(* CODESYS project CtaAppSupperheat_2.0.0.0.library
   Description: Überhitzungsregelungs- Library der CTA
   Version: 2.0.0.0
   Title: CtaAppSuperheat
   Author: SIS
   DocFormat: reStructuredText
   Placeholder: CtaAppSuperheat
   LanguageModelAttribute: qualified-access-only
   DefaultNamespace: CtaAppSuperheat
   CompiledLibraryCompatibilityVersion: CODESYS V3.5 SP16 Patch 3
   Company: CTA

Project tree, tasks and I/O mapping:
  libraries: Standard, 3.5.18.0 (System); CtaSysConfig, 2.0.0.0 (CTA); CtaVisSymbols, 2.0.0.0 (CTA); VisuDialogs, 3.5.16.20 (System); VisuSymbols, 4.5.0.0 (System); CtaAppReport, 2.0.0.0 (CTA); CtaAppDumper, 2.0.0.0 (CTA); CtaAppPid, 2.0.0.0 (CTA); CtaAppFilter, 1.0.0.0 (CTA); CtaAppBasic, 1.0.0.0 (CTA); CtaAppBmk, 2.0.0.0 (CTA); CtaAppInfluxLog, 1.0.0.1 (CTA); CtaVisHelp, 2.0.0.0 (CTA)
  40 Visualizations/
    Report/
      visualisation ReportIcon
      visualisation VIS_SUPERHEAT_REPORTS
    Settings/
      visualisation VIS_SUPERHEAT_SETTINGS
      visualisation VIS_SUPERHEAT_SETTINGS_BASE
    PopUp/
      visualisation PopUp
    VisSuperheat/
      visualisation visSuperheat
  00000000-0000-0000-0000-000000000000|D:\CoDeSys\LibrariesV3\trunk\Intern\CAA\CAA Template\3.4.0.0 draft\Placeholder.xml
  00000000-0000-0000-0000-000000000000|D:\CoDeSys\LibrariesV3\trunk\Intern\CAA\CAA Template\3.2.0.3 draft\Prefix.pdf
  00000000-0000-0000-0000-000000000000|D:\CoDeSys\LibrariesV3\trunk\Intern\CAA\CAA Template\3.5.2.0 draft\Placeholder.xml
  20 Structs/
    data type scParameter
    BASE/
      data type scBase
    InfluxDb/
      data type scInfluxDb
    LowSuperheat/
      data type scLowSuperheat
    MOP/
      data type scMOP
    Manual/
      data type scManual
  50 Images/
  10 Documenation/
    global variables VersionHistory
    global variables readMe
  21 Interface/
    interface ITF_Superheat: proAcknowleg, proAvailable, proLockDown, proIsError, proIsWarning, prorOnY, prorLowSuperheatValue, prorActÜberhitzung, prorSollÜberhitzung, p_scBase_fbxEnable, p_scBase_EnAlarmVentOffen, p_scBase_fbtDelayStartAlarm, p_scInfluxDb_fbxEnable, p_scLowSuperheat_fbrMin, p_scLowSuperheat_fbxEnable, p_scLowSuperheat_fbtDelayStartRegler, p_scLowSuperheat_fbrMax, p_scLowSuperheat_fbrMinÖffnung, p_scLowSuperheat_fbxEnableWarning, p_scLowSuperheat_fbxEnableAlarm, p_scLowSuperheat_fbtDelayStartAlarm, P_scLowSuperheat_fbrLowShAlarmValue, p_scMOP_fbxEnable, p_scMOP_fbxEnableWarning, p_scMOP_fbxEnableAlarm, p_scMOP_fbtDelayStartAlarm, p_scMOP_fbrMopSollwert, proRefTofbPidSuperheat, proRefTofbSuperheatDumper, proRefTofbPidMop, proRefTofbMopDumper, proITF_REPORTMANAGER
  11 Library Parameter/
  12 Konstanten/
    global variables GlobalKonstant
  60 Textlisten/
    text list Error
    text list Info
    text list Warnung
  13 Globale Variablen/
  text list GlobalTextList
  5ce3da45-db07-42e7-a21c-a00fff4ed8f6|C:\Users\sis\Downloads\dip-switch.svg
  5ce3da45-db07-42e7-a21c-a00fff4ed8f6|C:\Users\sis\Downloads\lightning-bolt-circle.svg
  30 Program Organization Units/
    function block fbSuperheat [ST]: actConfigFile, actReport, actTrendlog, actState, prorOnY, prorActÜberhitzung, prorLowSuperheatValue, prorSollÜberhitzung, proITF_REPORTMANAGER, proAcknowleg, proAvailable, proLockDown, proIsWarning, proIsError, p_scMOP_fbxEnable, p_scMOP_fbxEnableWarning, p_scMOP_fbxEnableAlarm, p_scMOP_fbtDelayStartAlarm, p_scMOP_fbrMopSollwert, p_scManual_fbxEnable, p_scManual_fbrManualValue, p_scInfluxDb_fbxEnable, p_scLowSuperheat_fbtDelayStartRegler, p_scLowSuperheat_fbrMin, p_scLowSuperheat_fbrMax, p_scLowSuperheat_fbrMinÖffnung, p_scLowSuperheat_fbxEnableWarning, p_scLowSuperheat_fbxEnableAlarm, p_scLowSuperheat_fbtDelayStartAlarm, p_scLowSuperheat_fbxEnable, P_scLowSuperheat_fbrLowShAlarmValue, p_scBase_fbxEnable, p_scBase_EnAlarmVentOffen, p_scBase_fbtDelayStartAlarm, proRefTofbPidSuperheat, proRefTofbSuperheatDumper, proRefTofbPidMop, proRefTofbMopDumper
    function fcProcentualReduction [ST]
  5ce3da45-db07-42e7-a21c-a00fff4ed8f6|C:\Users\sis\Downloads\sine-wave.svg
  5ce3da45-db07-42e7-a21c-a00fff4ed8f6|C:\Users\sis\Downloads\eye.svg
  5ce3da45-db07-42e7-a21c-a00fff4ed8f6|C:\Users\sis\Downloads\lan.svg
*)

// 20 Structs/scParameter
{attribute 'pack_mode' := '1'} 
TYPE scParameter :
	STRUCT
		scBase			: 	scBase;
		scLowSuperheat	:	scLowSuperheat;
		scMOP			:	scMOP;
		scManual		:	scManual;
		scInfluxDb		:	scInfluxDb;
	END_STRUCT
END_TYPE

// 20 Structs/BASE/scBase
TYPE scBase :
	STRUCT	
		fbxEnable				:	CtaSysConfig.fbBOOL;
		fbxEnAlarmVentOffen		:	CtaSysConfig.fbBOOL;
		fbtDelayStartAlarm		:	CtaSysConfig.fbTIME;		
	END_STRUCT
END_TYPE

// 20 Structs/InfluxDb/scInfluxDb
TYPE scInfluxDb :
	STRUCT		
		fbxEnable			:	CtaSysConfig.fbBOOL;
	END_STRUCT
END_TYPE

// 20 Structs/LowSuperheat/scLowSuperheat
TYPE scLowSuperheat :
	STRUCT
		fbxEnable				:	CtaSysConfig.fbBOOL;
		fbtDelayStartRegler		:	CtaSysConfig.fbTIME;
		fbrMin					:	CtaSysConfig.fbREAL;
		fbrMax					:	CtaSysConfig.fbREAL;
		fbrMinÖffnung			:	CtaSysConfig.fbREAL;
		fbxEnableWarning		:	CtaSysConfig.fbBOOL;
		fbxEnableAlarm			:	CtaSysConfig.fbBOOL;
		fbtDelayStartAlarm		:	CtaSysConfig.fbTIME;
		fbrLowShAlarmValue		:	CtaSysConfig.fbREAL;
	END_STRUCT
END_TYPE

// 20 Structs/MOP/scMOP
TYPE scMOP :
	STRUCT
		fbxEnable				:	CtaSysConfig.fbBOOL;
		fbxEnableWarning		:	CtaSysConfig.fbBOOL;
		fbxEnableAlarm			:	CtaSysConfig.fbBOOL;
		fbtDelayStartAlarm		:	CtaSysConfig.fbTIME;
		fbrMopSollwert			:	CtaSysConfig.fbREAL;
	END_STRUCT
END_TYPE

// 20 Structs/Manual/scManual
TYPE scManual :
	STRUCT
		fbxEnable		: CtaSysConfig.fbBOOL;
		fbrManualValue	: CtaSysConfig.fbREAL;
	END_STRUCT
END_TYPE

// 10 Documenation/VersionHistory
(* 

.. image:: ../../Images/CTA_Logo.jpg
   :align: right
   :width: 15% 

**Vorlage**   


============ =========== =========== ============================================
**Date**     **Version** **Author**  **Change**
------------ ----------- ----------- --------------------------------------------
04.03.2021   0.0.0.0     SIS         Vorlage erstellt

============ =========== =========== ============================================


*)
VAR_GLOBAL
    stInfo : STRING:= '0.0.0.0, Vorlage, CTA';
END_VAR

// 10 Documenation/readMe
(*

**ReadMe**
 
|	**Empfehlung**
|
|	Die Bibliothek CtaAppSuperheat dient der Überhitzungsregelung und errechnet den Stellwert für das elektronische Einspritzventil.
|	Instanzieren Sie den CtaAppSuperheat.fbSuperheat in ihrem Funktionsbaustein oder POU beispielsweise als fbSuperheatCtrl oder beliebig.
|	Deklarieren Sie die Struktur Variable welche als Parameter und zur ansteuerung dienen wie im Code beispiel.
|  
| *Beispiel* 

+-----------------------+---------------------------------------------------------------------------------------------------------------------------------------------------------------------------------------------------------------------------------------------------------------------------------------------------------------------------------------------------------------------------------------------------------------------------------------+
| Beschreibung          |  Code                                                                                                                                                                                                                                                                                                                                                                                                                                 |
+=======================+=======================================================================================================================================================================================================================================================================================================================================================================================================================================+
| Pou oder SmFb         | .. code-block:: codesys                                                                                                                                                                                                                                                                                                                                                                                                               |
|                       |                                                                                                                                                                                                                                                                                                                                                                                                                                       |
|                       |	// Deklaration als VAR im POU oder dem selbsterstellten Funktionsbaustein                                                                                                                                                                                                                                                                                                                                                       	|
|                       |   VAR   																																																																																																								|
|						|	    (*Überhitzungsregelung*)																																																		 																																																|
|						|		fbSuperheatCtrl			: CtaAppSuperheat.fbSuperheat;                                                                                                                                                                                                                                                                                                                                                             				|
|						|																																																																																																										|
+-----------------------+---------------------------------------------------------------------------------------------------------------------------------------------------------------------------------------------------------------------------------------------------------------------------------------------------------------------------------------------------------------------------------------------------------------------------------------+
| Code für Init         | .. code-block:: codesys                                                                                                                                                                                                                                                                                                                                                                                                               |
|                       |   																																																																																																									|
| 						|	// Kopieren des nachfolgenden Codes in eine Action zur Initialisierung der Parameter. Zum Beispiel actConfig.																																																																														|
|                       |	{region "Überhitzungsregelung																																																																																																		|
|						|		(*Base*)                                                                                                                                                                                                                                                                                                                                                                                                   						|
|						|		fbSuperheatCtrl.scParameter.scBase.fbxEnable						(_wertInit :=	 TRUE														);		//P1 Überhitzungsregelung aktiv / inaktiv																																																								|
|						|		fbSuperheatCtrl.scParameter.scBase.fbrStartÖffnung					(_wertInit :=	   20		, _minInit :=			, _maxInit :=			);		//P2 Startöffnung des Ventils																																																											|
|						|		fbSuperheatCtrl.scParameter.scBase.fbtDelayStartRegler				(_wertInit :=	T#10s		, _minInit :=			, _maxInit :=			);		//P3 Startverzögerung der Regelung																																																										|
|						|		fbSuperheatCtrl.scParameter.scBase.fbxEnAlarmVentOffen				(_wertInit :=	FALSE														);		//P4 Alarm bei 100% geöffnetem Ventil aktiv / inaktiv																																																					|
|						|		fbSuperheatCtrl.scParameter.scBase.fbtDelayStartAlarm				(_wertInit :=	 T#0S		, _minInit :=			, _maxInit :=			);		//P5 Alarmverzögerung 																																																													|
|						|																																																																																																										|
|						|		(*Superheat PID*)																																																																																																				|
|						|		fbSuperheatCtrl.fbPidSuperheat.scParameter.fbrBand					(_wertInit :=	   15		, _minInit :=			, _maxInit :=			);		//P6  Superheat PID - Band																																																												|
|						|		fbSuperheatCtrl.fbPidSuperheat.scParameter.fbrDeadBand				(_wertInit :=	 0.10		, _minInit :=			, _maxInit :=			);		//P7  Superheat PID - Totband																																																											|
|						|		fbSuperheatCtrl.fbPidSuperheat.scParameter.fbrTn					(_wertInit :=	   25		, _minInit :=			, _maxInit :=			);		//P8  Superheat PID - I Anteil																																																											|
|						|		fbSuperheatCtrl.fbPidSuperheat.scParameter.fbrTv					(_wertInit :=	    2		, _minInit :=			, _maxInit :=			);		//P9  Superheat PID - D Anteil																																																											|
|						|		fbSuperheatCtrl.fbPidSuperheat.scParameter.fbxEnTrendlog			(_wertInit :=	FALSE														);		//P10 Superheat PID - Trendaufzeichnung																																																									|
|						|		fbSuperheatCtrl.fbPidSuperheat.scParameter.fbxInvert				(_wertInit :=	FALSE														);		//P11 Superheat PID - Invrtierung																																																										|
|						|																																																																																																										|
|						|		(*Superheat Dumper*)																																																																																																			|
|						|		fbSuperheatCtrl.fbSuperheatDumper.scParameter.fbrBand				(_wertInit :=	  100		, _minInit :=			, _maxInit :=			);		//P12 Superheat Dumper - Band																																																											|
|						|		fbSuperheatCtrl.fbSuperheatDumper.scParameter.fbrTup				(_wertInit :=	   10		, _minInit :=			, _maxInit :=			);		//P13 Superheat Dumper - Zuschaltzeit																																																									|
|						|		fbSuperheatCtrl.fbSuperheatDumper.scParameter.fbrTdown				(_wertInit :=	    1		, _minInit :=			, _maxInit :=			);		//P14 Superheat Dumper - Wegschaltzeit																																																									|
|						|		fbSuperheatCtrl.fbSuperheatDumper.scParameter.fbxInExpOut			(_wertInit :=	FALSE														);		//P15 Superheat Dumper - In = Out annahme																																																								|
|						|																																																																																																										|
|						|		(*Low Superheat*)																																																																																																				|
|						|		fbSuperheatCtrl.scParameter.scLowSuperheat.fbxEnable				(_wertInit :=	 TRUE														);		//P16 LowSuperheat aktiv / inaktiv																																																										|
|						|		fbSuperheatCtrl.scParameter.scLowSuperheat.fbrMin					(_wertInit :=	  2.0		, _minInit :=			, _maxInit :=			);		//P17 LowSuperheat Minimalwert																																																											|
|						|		fbSuperheatCtrl.scParameter.scLowSuperheat.fbrMax					(_wertInit :=	  3.0		, _minInit :=			, _maxInit :=			);		//P18 LowSuperheat Maximalwert																																																											|
|						|		fbSuperheatCtrl.scParameter.scLowSuperheat.fbrMinÖffnung			(_wertInit :=	 	0		, _minInit :=			, _maxInit :=			);		//P19 LowSuperheat Minimalöffnung																																																										|
|						|		fbSuperheatCtrl.scParameter.scLowSuperheat.fbtDelayStartRegler		(_wertInit :=	T#30s		, _minInit :=			, _maxInit :=			);		//P20 LowSuperheat Regler Startverzögerung																																																								|
|						|		fbSuperheatCtrl.scParameter.scLowSuperheat.fbxEnableWarning			(_wertInit :=	 TRUE														);		//P21 LowSuperheat Warnung aktiv / inaktiv																																																								|
|						|		fbSuperheatCtrl.scParameter.scLowSuperheat.fbxEnableAlarm			(_wertInit :=	 TRUE														);		//P22 LowSuperheat Alarm aktiv / inaktiv																																																								|
|						|		fbSuperheatCtrl.scParameter.scLowSuperheat.fbtDelayStartAlarm		(_wertInit :=	T#30s		, _minInit :=			, _maxInit :=			);		//P23 LowSuperheat Alarmverzögerung																																																										|
|						|																																																																																																										|
|						|		(*MOP*)																																																																																																							|
|						|		fbSuperheatCtrl.scParameter.scMOP.fbxEnable							(_wertInit :=	 TRUE														);		//P24 MOP aktiv / inaktiv																																																												|
|						|		fbSuperheatCtrl.scParameter.scMOP.fbxEnableWarning					(_wertInit :=	 TRUE														);		//P25 MOP Warnung aktiv / inaktiv																																																										|
|						|		fbSuperheatCtrl.scParameter.scMOP.fbxEnableAlarm					(_wertInit :=	 TRUE														);		//P26 MOP Alarm aktiv / inaktiv																																																											|
|						|		fbSuperheatCtrl.scParameter.scMOP.fbtDelayStartAlarm				(_wertInit :=	T#10s		, _minInit :=			, _maxInit :=			);		//P27 MOP Alarmverzögerung																																																												|
|						|																																																																																																										|
|						|		(*MOP Leistungsreduktion*)																																																																																																		|
|						|		fbSuperheatCtrl.fbMopLeistungsreduktion.scParameter.fbxEn			(_wertInit :=	 TRUE														);		//P28 MOP Leistungsreduktion aktiv / inaktiv 																																																							|
|						|		fbSuperheatCtrl.fbMopLeistungsreduktion.scParameter.fbtStartTime	(_wertInit :=	 T#1m		, _minInit :=			, _maxInit :=			);		//P29 MOP Leistungsreduktion Regler Startverzögerung																																																					|
|						|		fbSuperheatCtrl.fbMopLeistungsreduktion.scParameter.fbtRunTime		(_wertInit :=	 T#1m		, _minInit :=			, _maxInit :=			);		//P30 MOP Leistungsreduktion Regler Betriebsverzögerung																																																					|
|						|		fbSuperheatCtrl.fbMopLeistungsreduktion.scParameter.fbrSoll			(_wertInit :=	   10		, _minInit :=			, _maxInit :=			);		//P31 MOP Leistungsreduktion Sollwert																																																									|
|						|		fbSuperheatCtrl.fbMopLeistungsreduktion.scParameter.fbrCounter		(_wertInit :=	 	5		, _minInit :=			, _maxInit :=			);		//P32 MOP Leistungsreduktion Weg- / Zuschaltungwert																																																						|
|						|		fbSuperheatCtrl.fbMopLeistungsreduktion.scParameter.fbxEnTrendLog	(_wertInit :=	 TRUE														);		//P33 MOP Leistungsreduktion Trendaufzeichnung																																																							|
|						|																																																																																																										|
|						|		(*MOP Dumper*)																																																																																																					|
|						|		fbSuperheatCtrl.fbMopDumper.scParameter.fbrBand						(_wertInit :=	  0.0		, _minInit :=			, _maxInit :=			);		//P34 MOP Dumper - Band																																																													|
|						|		fbSuperheatCtrl.fbMopDumper.scParameter.fbrTdown					(_wertInit :=	 0.10		, _minInit :=			, _maxInit :=			);		//P35 MOP Dumper - Zuschaltzeit																																																											|
|						|		fbSuperheatCtrl.fbMopDumper.scParameter.fbrTup						(_wertInit :=	 0.10		, _minInit :=			, _maxInit :=			);		//P36 MOP Dumper - Wegschaltzeit																																																										|
|						|		fbSuperheatCtrl.fbMopDumper.scParameter.fbxInExpOut					(_wertInit :=	FALSE														);		//P37 MOP In = Out annahme																																																												|
|						|																																																																																																										|
|						|		(*Manual*)																																																																																																						|
|						|		fbSuperheatCtrl.scParameter.scManual.fbxEnable						(_wertInit :=	FALSE														);		//P38 Manuelle Übersteuerung aktivieren / deaktivieren																																																					|
|						|		fbSuperheatCtrl.scParameter.scManual.fbrManualValue					(_wertInit :=	 	0		, _minInit :=			, _maxInit :=			);		//P39 Manueller Ventilstellwert																																																											|
|						|																																																																																																										|
|						|		(*Trendlog*)																																																																																																					|
|						|		fbSuperheatCtrl.scParameter.scInfluxDb.fbxEnable					(_wertInit :=	 TRUE														);		//P40 Überhitzungsregelung Trendaufzeichnung																																																							|
|						|	{endregion}                                                                                                                                                      																																																																	|
+-----------------------+---------------------------------------------------------------------------------------------------------------------------------------------------------------------------------------------------------------------------------------------------------------------------------------------------------------------------------------------------------------------------------------------------------------------------------------+
*)                                                                                                                                                                                                                                                                                                                                                                                                                                                               
 VAR_GLOBAL                                                                                                                                                                                                                                                                                                                                                                                                                                                      
    xReadMeDone              :   BOOL;                                                                                                                                                                                                                                                                                                                                                                                                                           
END_VAR

// 12 Konstanten/GlobalKonstant
{attribute 'qualified_only'}
VAR_GLOBAL
	stReportTextListError   : CtaAppReport.stReportTextList := 'CtaAppSuperheat.Error';
	stReportTextListWarning : CtaAppReport.stReportTextList := 'CtaAppSuperheat.Warnung';
	stReportTextListInfo    : CtaAppReport.stReportTextList := 'CtaAppSuperheat.Info';	
END_VAR

// 30 Program Organization Units/fbSuperheat
FUNCTION_BLOCK fbSuperheat IMPLEMENTS ITF_Superheat
VAR_INPUT
	
	//Überhitzungsregler   
    xRelease						: BOOL;	// Freigabe Regulierung, Beispiel Freigabe Verdichter
    rSollÜberhitzung				: REAL;	// Sollwert Überhitzung
    rKorrekturÜberhizungssollwert	: REAL;	// Korrektur von Sollwert, Schiebungswert muss aussen gemacht werden
    rActSauggastemperatur			: REAL;
    rActVerdampfungstemperatur		: REAL;
	ITF_BMK							: CtaAppBmk.ITF_BMK;
	
END_VAR
VAR_OUTPUT
	 rOnY							: REAL;	// Aktueller Stellwert für Expansionsventil
END_VAR
VAR
	(* Internal States *) 
	scEWI							: CtaAppReport.scReportNr;
	_xIsWarning						: BOOL;
	xIsWarning						: BOOL;
	_xIsError						: BOOL;
	xIsError						: BOOL;
	xisEnabled						: BOOL;
		
	(* Temps and Helpers *)
	rLowSuperheatScaled				: REAL;
	xConfigError					: BOOL;
	
	(* Bausteine Superheat *)	
	fbPidSuperheat					: CtaAppPid.fbPid;
	fbSuperheatDumper				: CtaAppDumper.fbDumper;
	
	(* Bausteine Low Superheat *)
	fbLowSuperheatDelay				: Standard.TON;
	fbLowSuperheatSetReset			: Standard.RS;
	fbLowSuperheatFilter			: CtaAppFilter.fbImpulsFilter;
	
	(* Bausteine MOP *)
	fbPidMop						: CtaAppPid.fbPid;
	fbMopDumper						: CtaAppDumper.fbDumper;
	
	(* Reporting *) 
	fbReportManager			    	: CtaAppReport.fbReportManager;      
    difor					    	: DINT;                                                                    
    ayErrorReporter					: ARRAY[1..5] OF CtaAppReport.fbReporter;
	ayWarningReporter				: ARRAY[1..2] OF CtaAppReport.fbReporter;
	
	(* Trendlogs *)
	fbTrendxOn						:	CtaAppInfluxLog.FB_LOG_NODE_BOOL;
	fbTrendrOny						:	CtaAppInfluxLog.FB_LOG_NODE_REAL;
	fbTrendxWarning					:	CtaAppInfluxLog.FB_LOG_NODE_BOOL;
	fbTrendxError					:	CtaAppInfluxLog.FB_LOG_NODE_BOOL;
	(* ConfigFile *)
	fbConfigfile					: CtaSysConfig.fbConfigFile;
	scParameter						: scParameter;
END_VAR

actConfigFile();

IF xIsEnabled AND NOT xConfigError THEN
	
	(* Superheat *)
	
		// PID
		fbPidSuperheat(	xEn 					:=	xRelease,
						rAct 					:=	rActSauggastemperatur - rActVerdampfungstemperatur,
						rSoll 					:=	rSollÜberhitzung + rKorrekturÜberhizungssollwert,
						stPhysikalischeEinheit 	:=	'°c');
						
		// Skalierung 			
		fbSuperheatDumper.rSoll :=  CtaAppBasic.fcScale(rIn 	:= fbPidSuperheat.rY,
														rMin 	:=	-100,
														rMax 	:=	 100,
														rOutMin	:=	   0,
														rOutMax	:=   100);
		// Dämpfung des skalierten Wertes												
		fbSuperheatDumper(xEn := TRUE);				
	
	(* Low Superheat *)
		// Skalierung
		rLowSuperheatScaled := MAX (0 , CtaAppBasic.fcScale(rIn 	:= fbPidSuperheat.rAct,
															rMin 	:= scParameter.scLowSuperheat.fbrMin.proValue,
															rMax 	:= scParameter.scLowSuperheat.fbrMax.proValue,
															rOutMin := 100 - scParameter.scLowSuperheat.fbrMinÖffnung.proValue,
															rOutMax := 0));
		
		// Verzögerung der Regelung
		fbLowSuperheatDelay(IN :=	xRelease 										AND
									(rLowSuperheatScaled > 0) 						AND 
								 	NOT fbLowSuperheatSetReset.Q1 					AND
								  	scParameter.scLowSuperheat.fbxEnable.proValue,
							PT := 	scParameter.scLowSuperheat.fbtDelayStartRegler.proValue);
							
		// Set Reset					
		fbLowSuperheatSetReset(	SET 	:= fbLowSuperheatDelay.Q ,
								RESET1 	:= NOT xRelease);
		
		// Wert für prozentuale Reduktion LowSuperheat				
		IF fbLowSuperheatSetReset.Q1 THEN
			fbLowSuperheatFilter.rIn := rLowSuperheatScaled;
		ELSE
			fbLowSuperheatFilter.rIn := 0;
		END_IF
		
		// Filterung des Wertes
		fbLowSuperheatFilter(rFilter := 10.0);
		
		// LowSuperheat reporting in der Aktion actReport realisiert
	
	(* MOP *)
		// Leistungreduktion
		fbPidMop(	xEn 					:= xRelease AND scParameter.scMOP.fbxEnable.proValue,
					rAct 					:= rActVerdampfungstemperatur,
					rSoll 					:= scParameter.scMOP.fbrMopSollwert.proValue,
					stPhysikalischeEinheit 	:= '°c'  );
								
		// Dämpfung des MOP- Wertes
		fbMopDumper(xEn 	:= xRelease AND scParameter.scMOP.fbxEnable.proValue,
					rSoll 	:= LIMIT(0,fbPidMop.rY,100));
		
		// MOP Reporting in der Aktion actReport realisiert
	
	(* Stellwert *)
	IF xRelease THEN
		// Ausgang mit prozentualer Reduktion beschalten
		fcProcentualReduction(	rLAkt 	:= fbSuperheatDumper.rY,
								rLR1	:= fbLowSuperheatFilter.rOut,
								rLR2	:= fbMopDumper.rY,
								rOut	=> rOnY);		
	ELSE
		rOnY := 0;	
	END_IF	
	
	// Reports
	IF __QUERYINTERFACE(ITF_BMK,ITF_BMK)THEN
		actReport();
	END_IF
ELSE
	// Stellwertreporting in der Atkion actReport realisiert
	rOnY := 0;
	
	// Konfigurationsfehler
	IF xConfigError THEN
		IF __QUERYINTERFACE(ITF_BMK,ITF_BMK)THEN
			actReport();
		END_IF
	END_IF	
END_IF

// Status
actState();
// Trends
IF __QUERYINTERFACE(ITF_BMK,ITF_BMK) THEN
	actTrendlog();
END_IF

ACTION actConfigFile:
fbConfigfile();

(* Basisparameter *)
scParameter.scBase.fbxEnable					(_usiParaNr :=  1, ItfConfigFb := fbConfigFile);
scParameter.scBase.fbxEnAlarmVentOffen 			(_usiParaNr :=  4, ItfConfigFb := fbConfigFile);
scParameter.scBase.fbtDelayStartAlarm			(_usiParaNr :=  5, ItfConfigFb := fbConfigFile);
(* Low Superheat *)
scParameter.scLowSuperheat.fbxEnable			(_usiParaNr :=  6, ItfConfigFb := fbConfigFile);
scParameter.scLowSuperheat.fbtDelayStartRegler	(_usiParaNr :=  7, ItfConfigFb := fbConfigFile);
scParameter.scLowSuperheat.fbrMin				(_usiParaNr :=  8, ItfConfigFb := fbConfigFile);
scParameter.scLowSuperheat.fbrMax				(_usiParaNr :=  9, ItfConfigFb := fbConfigFile);
scParameter.scLowSuperheat.fbrMinÖffnung		(_usiParaNr := 10, ItfConfigFb := fbConfigFile);
scParameter.scLowSuperheat.fbxEnableWarning		(_usiParaNr := 11, ItfConfigFb := fbConfigFile);
scParameter.scLowSuperheat.fbxEnableAlarm		(_usiParaNr := 12, ItfConfigFb := fbConfigFile);
scParameter.scLowSuperheat.fbtDelayStartAlarm	(_usiParaNr := 13, ItfConfigFb := fbConfigFile);
(* MOP Regler *)
scParameter.scMOP.fbxEnable						(_usiParaNr := 14, ItfConfigFb := fbConfigFile);
scParameter.scMOP.fbxEnableWarning				(_usiParaNr := 15, ItfConfigFb := fbConfigFile);
scParameter.scMOP.fbxEnableAlarm				(_usiParaNr := 16, ItfConfigFb := fbConfigFile);
scParameter.scMOP.fbtDelayStartAlarm			(_usiParaNr := 17, ItfConfigFb := fbConfigFile);
scParameter.scMOP.fbrMopSollwert				(_usiParaNr := 18, ItfConfigFb := fbConfigFile);
(* Trendlog *)
scParameter.scInfluxDb.fbxEnable				(_usiParaNr := 19, ItfConfigFb := fbConfigFile);

scParameter.scLowSuperheat.fbrLowShAlarmValue	(_usiParaNr := 20, ItfConfigFb := fbConfigFile);

xConfigError := fbConfigFile.xError;
END_ACTION

ACTION actReport:
(* EWI Manager *)
fbReportManager(	stErrorInitReportTextListIn		:=	ADR(GlobalKonstant.stReportTextListError),
					stWarningInitReportTextListIn	:=	ADR(GlobalKonstant.stReportTextListWarning),
					stInfoInitReportTextListIn		:=	ADR(GlobalKonstant.stReportTextListInfo),
					scReportNr						:=	scEWI);
					
(* Errors *)                        
        (* Meldung Error Low Superheat *)
        ayErrorReporter[1].proPrio  := 3;
        ayErrorReporter[1].metReport(     		xSetReportIn					:= xRelease AND 
																				   (rLowSuperheatScaled > 0) AND 
																				   scParameter.scLowSuperheat.fbxEnable.proValue AND
																				   scParameter.scLowSuperheat.fbxEnableAlarm.proValue,
												iReportID						:= 1,
												enReportTypeIn					:= CtaAppReport.enReportType.Error,  
												enReportAcknowledgeTypeIn   	:= CtaAppReport.enReportacknowledgeType.Quit,
												tDelay							:= scParameter.scLowSuperheat.fbtDelayStartAlarm.proValue, 
												ITF_BMK_IN						:= ITF_BMK,			              
												pstReportTextListIn				:= ADR(GlobalKonstant.stReportTextListError),
												stOptionalReportText		    := '',   
												iRetryTilReportLock 		    := 0, 
												xResetCount         		    := FALSE,  
												tReset						    := T#24H); 

		(* Meldung Error MOP *)
        ayErrorReporter[2].proPrio  := 3;
        ayErrorReporter[2].metReport(     		xSetReportIn					:= xRelease 			AND
																				   fbMopDumper.rY > 0 	AND 
																				   scParameter.scMOP.fbxEnableAlarm.proValue,
												iReportID						:= 2,
												enReportTypeIn					:= CtaAppReport.enReportType.Error,  
												enReportAcknowledgeTypeIn   	:= CtaAppReport.enReportacknowledgeType.Quit,
												tDelay							:= scParameter.scMOP.fbtDelayStartAlarm.proValue, 
												ITF_BMK_IN						:= ITF_BMK,			              
												pstReportTextListIn				:= ADR(GlobalKonstant.stReportTextListError),
												stOptionalReportText		    := '',   
												iRetryTilReportLock 		    := 0, 
												xResetCount         		    := FALSE,  
												tReset						    := T#24H);

		(* Meldung Error Ventil *)
        ayErrorReporter[3].proPrio  := 3;
        ayErrorReporter[3].metReport(     		xSetReportIn					:= (rOnY > 99.9) AND
																				   scParameter.scBase.fbxEnAlarmVentOffen.proValue,
												iReportID						:= 3,
												enReportTypeIn					:= CtaAppReport.enReportType.Error,  
												enReportAcknowledgeTypeIn   	:= CtaAppReport.enReportacknowledgeType.Quit,
												tDelay							:= scParameter.scBase.fbtDelayStartAlarm.proValue, 
												ITF_BMK_IN						:= ITF_BMK,			              
												pstReportTextListIn				:= ADR(GlobalKonstant.stReportTextListError),
												stOptionalReportText		    := '',   
												iRetryTilReportLock 		    := 0, 
												xResetCount         		    := FALSE,  
												tReset						    := T#24H);		
												
		(* Meldung Configerror *)
        ayErrorReporter[4].proPrio  := 1;
        ayErrorReporter[4].metReport(     		xSetReportIn					:= xConfigError,
												iReportID						:= 4,
												enReportTypeIn					:= CtaAppReport.enReportType.Error,  
												enReportAcknowledgeTypeIn   	:= CtaAppReport.enReportacknowledgeType.Quit,
												tDelay							:= scParameter.scBase.fbtDelayStartAlarm.proValue, 
												ITF_BMK_IN						:= ITF_BMK,			              
												pstReportTextListIn				:= ADR(GlobalKonstant.stReportTextListError),
												stOptionalReportText		    := '',   
												iRetryTilReportLock 		    := 0, 
												xResetCount         		    := FALSE,  
												tReset						    := T#24H);	

        (* Meldung Error Low Superheat *)
        ayErrorReporter[5].proPrio  := 1;
        ayErrorReporter[5].metReport(     		xSetReportIn					:= xRelease AND rActSauggastemperatur - rActVerdampfungstemperatur < scParameter.scLowSuperheat.fbrLowShAlarmValue.proValue,
												iReportID						:= 5,
												enReportTypeIn					:= CtaAppReport.enReportType.Error,  
												enReportAcknowledgeTypeIn   	:= CtaAppReport.enReportacknowledgeType.Quit,
												tDelay							:= T#1.5S, 
												ITF_BMK_IN						:= ITF_BMK,			              
												pstReportTextListIn				:= ADR(GlobalKonstant.stReportTextListError),
												stOptionalReportText		    := '',   
												iRetryTilReportLock 		    := 0, 
												xResetCount         		    := FALSE,  
												tReset						    := T#24H); 
												
(* Warnungen *)      
        (* Warnung Low Superheat *)      
        ayWarningReporter[1].proPrio := 2;
        ayWarningReporter[1].metReport(			xSetReportIn					:= xRelease AND 
																				   (rLowSuperheatScaled > 0) AND
																				   scParameter.scLowSuperheat.fbxEnable.proValue AND
																				   scParameter.scLowSuperheat.fbxEnableWarning.proValue,
												iReportID						:= 1,
												enReportTypeIn					:= CtaAppReport.enReportType.Warning,  
												enReportAcknowledgeTypeIn   	:= CtaAppReport.enReportAcknowledgeType.Auto,
												tDelay							:= T#0S, 
												ITF_BMK_IN						:= ITF_BMK,			              
												pstReportTextListIn				:= ADR(GlobalKonstant.stReportTextListWarning),
												stOptionalReportText		    := '',   
												iRetryTilReportLock 		    := 0, 
												xResetCount         		    := FALSE,  
												tReset						    := T#24H);  
		(* Warnung MOP *)      
        ayWarningReporter[2].proPrio := 2;
        ayWarningReporter[2].metReport(			xSetReportIn					:= xRelease 			AND 
																				   fbMopDumper.rY > 0	AND
																				   scParameter.scMOP.fbxEnableWarning.proValue,
												iReportID						:= 2,
												enReportTypeIn					:= CtaAppReport.enReportType.Warning,  
												enReportAcknowledgeTypeIn   	:= CtaAppReport.enReportAcknowledgeType.Auto,
												tDelay							:= T#0S, 
												ITF_BMK_IN						:= ITF_BMK,			              
												pstReportTextListIn				:= ADR(GlobalKonstant.stReportTextListWarning),
												stOptionalReportText		    := '',   
												iRetryTilReportLock 		    := 0, 
												xResetCount         		    := FALSE,  
												tReset						    := T#24H);            
												
(* Sync Reports *)                                         
FOR difor := LOWER_BOUND(ayErrorReporter,1) TO UPPER_BOUND(ayErrorReporter,1) DO
	fbReportManager.metSyncReporter(ayErrorReporter[difor]);	
END_FOR;
FOR difor := LOWER_BOUND(ayWarningReporter,1) TO UPPER_BOUND(ayWarningReporter,1) DO
	fbReportManager.metSyncReporter(ayWarningReporter[difor]);	
END_FOR;
                                                                             
_xIsError   := scEWI.iError <> 0;
_xIsWarning := scEWI.iWarning <> 0;
END_ACTION

ACTION actTrendlog:
(* Schaltbefehl *)
fbTrendxOn.ENABLE			:=	scParameter.scBase.fbxEnable.proValue AND
								scParameter.scInfluxDb.fbxEnable.proValue;
fbTrendxOn.KEY 				:=	CONCAT(ITF_BMK.proGetObjectId,'_Supperheat_xOn');
fbTrendxOn.SET_VALUE		:=	xRelease;

(* Stellwert *)
fbTrendrOny.ENABLE			:=	scParameter.scBase.fbxEnable.proValue AND
								scParameter.scInfluxDb.fbxEnable.proValue;
fbTrendrOny.KEY 			:=	CONCAT(ITF_BMK.proGetObjectId,'_Supperheat_rOnY');
fbTrendrOny.SET_VALUE		:=  rOnY;

(* Warnung *)
fbTrendxWarning.ENABLE		:=	scParameter.scBase.fbxEnable.proValue AND
								scParameter.scInfluxDb.fbxEnable.proValue;
fbTrendxWarning.KEY 		:=	CONCAT(ITF_BMK.proGetObjectId,'_Supperheat_xWarning');
fbTrendxWarning.SET_VALUE	:=  xIsWarning;

(* Fehler *)
fbTrendxError.ENABLE		:=	scParameter.scBase.fbxEnable.proValue AND
								scParameter.scInfluxDb.fbxEnable.proValue;
fbTrendxError.KEY 			:=	CONCAT(ITF_BMK.proGetObjectId,'_Supperheat_xError');
fbTrendxError.SET_VALUE		:=  xIsError;
END_ACTION

ACTION actState:
xisEnabled  := scParameter.scBase.fbxEnable.proValue;
xIsWarning 	:= _xIsWarning;
xIsError	:= _xIsError;
END_ACTION

PROPERTY prorOnY : REAL
GET
prorOnY := rOnY;
END_GET
END_PROPERTY

PROPERTY prorActÜberhitzung : REAL
GET
prorActÜberhitzung := fbPidSuperheat.rAct;
END_GET
END_PROPERTY

PROPERTY prorLowSuperheatValue : REAL
GET
prorLowSuperheatValue := fbLowSuperheatFilter.rOut;
END_GET
END_PROPERTY

PROPERTY prorSollÜberhitzung : REAL
GET
prorSollÜberhitzung := fbPidSuperheat.rSoll;
END_GET
END_PROPERTY

PROPERTY proITF_REPORTMANAGER : CtaAppReport.ITF_REPORTMANAGER
GET
proITF_REPORTMANAGER := fbReportManager;
END_GET
END_PROPERTY

{attribute 'monitoring' := 'variable'}
PROPERTY proAcknowleg : BOOL
GET
proAcknowleg := xRelease AND NOT xIsError;
END_GET
END_PROPERTY

{attribute 'monitoring' := 'variable'}
PROPERTY proAvailable : BOOL
GET
proAvailable := scParameter.scBase.fbxEnable.proValue AND NOT xIsError;
END_GET
END_PROPERTY

{attribute 'monitoring' := 'variable'}
PROPERTY proLockDown : BOOL
GET
proLockDown := xIsError;
END_GET
END_PROPERTY

PROPERTY proIsWarning : BOOL
GET
proIsWarning := xIsWarning;
END_GET
END_PROPERTY

PROPERTY proIsError : BOOL
GET
proIsError := xIsError;
END_GET
END_PROPERTY

PROPERTY p_scMOP_fbxEnable : CtaSysConfig.ITF_DATATYPE
GET
p_scMOP_fbxEnable := scParameter.scMOP.fbxEnable;
END_GET
END_PROPERTY

PROPERTY p_scMOP_fbxEnableWarning : CtaSysConfig.ITF_DATATYPE
GET
p_scMOP_fbxEnableWarning := scParameter.scMOP.fbxEnableWarning;
END_GET
END_PROPERTY

PROPERTY p_scMOP_fbxEnableAlarm : CtaSysConfig.ITF_DATATYPE
GET
p_scMOP_fbxEnableAlarm := scParameter.scMOP.fbxEnableAlarm;
END_GET
END_PROPERTY

PROPERTY p_scMOP_fbtDelayStartAlarm : CtaSysConfig.ITF_DATATYPE
GET
p_scMOP_fbtDelayStartAlarm := scParameter.scMOP.fbtDelayStartAlarm;
END_GET
END_PROPERTY

PROPERTY p_scMOP_fbrMopSollwert : CtaSysConfig.ITF_DATATYPE
GET
p_scMOP_fbrMopSollwert := scParameter.scMOP.fbrMopSollwert;
END_GET
END_PROPERTY

PROPERTY p_scManual_fbxEnable : CtaSysConfig.ITF_DATATYPE
GET
p_scManual_fbxEnable := scParameter.scManual.fbxEnable;
END_GET
END_PROPERTY

PROPERTY p_scManual_fbrManualValue : CtaSysConfig.ITF_DATATYPE
GET
p_scManual_fbrManualValue := scParameter.scManual.fbrManualValue;
END_GET
END_PROPERTY

PROPERTY p_scInfluxDb_fbxEnable : CtaSysConfig.ITF_DATATYPE
GET
p_scInfluxDb_fbxEnable := scParameter.scInfluxDb.fbxEnable;
END_GET
END_PROPERTY

PROPERTY p_scLowSuperheat_fbtDelayStartRegler : CtaSysConfig.ITF_DATATYPE
GET
p_scLowSuperheat_fbtDelayStartRegler := scParameter.scLowSuperheat.fbtDelayStartRegler;
END_GET
END_PROPERTY

PROPERTY p_scLowSuperheat_fbrMin : CtaSysConfig.ITF_DATATYPE
GET
p_scLowSuperheat_fbrMin := scParameter.scLowSuperheat.fbrMin;
END_GET
END_PROPERTY

PROPERTY p_scLowSuperheat_fbrMax : CtaSysConfig.ITF_DATATYPE
GET
p_scLowSuperheat_fbrMax := scParameter.scLowSuperheat.fbrMax;
END_GET
END_PROPERTY

PROPERTY p_scLowSuperheat_fbrMinÖffnung : CtaSysConfig.ITF_DATATYPE
GET
p_scLowSuperheat_fbrMinÖffnung := scParameter.scLowSuperheat.fbrMinÖffnung;
END_GET
END_PROPERTY

PROPERTY p_scLowSuperheat_fbxEnableWarning : CtaSysConfig.ITF_DATATYPE
GET
p_scLowSuperheat_fbxEnableWarning := scParameter.scLowSuperheat.fbxEnableWarning;
END_GET
END_PROPERTY

PROPERTY p_scLowSuperheat_fbxEnableAlarm : CtaSysConfig.ITF_DATATYPE
GET
p_scLowSuperheat_fbxEnableAlarm := scParameter.scLowSuperheat.fbxEnableAlarm;
END_GET
END_PROPERTY

PROPERTY p_scLowSuperheat_fbtDelayStartAlarm : CtaSysConfig.ITF_DATATYPE
GET
p_scLowSuperheat_fbtDelayStartAlarm := scParameter.scLowSuperheat.fbtDelayStartAlarm;
END_GET
END_PROPERTY

PROPERTY p_scLowSuperheat_fbxEnable : CtaSysConfig.ITF_DATATYPE
GET
p_scLowSuperheat_fbxEnable := scParameter.scLowSuperheat.fbxEnable;
END_GET
END_PROPERTY

PROPERTY P_scLowSuperheat_fbrLowShAlarmValue : CtaSysConfig.ITF_REAL
GET
P_scLowSuperheat_fbrLowShAlarmValue := scParameter.scLowSuperheat.fbrLowShAlarmValue;
END_GET
END_PROPERTY

PROPERTY p_scBase_fbxEnable : CtaSysConfig.ITF_DATATYPE
GET
p_scBase_fbxEnable := scParameter.scBase.fbxEnable;
END_GET
END_PROPERTY

PROPERTY p_scBase_EnAlarmVentOffen : CtaSysConfig.ITF_DATATYPE
GET
p_scBase_EnAlarmVentOffen := scParameter.scBase.fbxEnAlarmVentOffen;
END_GET
END_PROPERTY

PROPERTY p_scBase_fbtDelayStartAlarm : CtaSysConfig.ITF_DATATYPE
GET
p_scBase_fbtDelayStartAlarm := scParameter.scBase.fbtDelayStartAlarm;
END_GET
END_PROPERTY

PROPERTY proRefTofbPidSuperheat : REFERENCE TO CtaAppPid.fbPid
GET
proRefTofbPidSuperheat REF= fbPidSuperheat;
END_GET
END_PROPERTY

PROPERTY proRefTofbSuperheatDumper : REFERENCE TO CtaAppDumper.fbDumper
GET
proRefTofbSuperheatDumper REF= fbSuperheatDumper;
END_GET
END_PROPERTY

PROPERTY proRefTofbPidMop: REFERENCE TO CtaAppPid.fbPid
GET
proRefTofbPidMop REF= fbPidMop;
END_GET
END_PROPERTY

PROPERTY proRefTofbMopDumper : REFERENCE TO CtaAppDumper.fbDumper
GET
proRefTofbMopDumper REF= fbMopDumper;
END_GET
END_PROPERTY

END_FUNCTION_BLOCK

// 30 Program Organization Units/fcProcentualReduction
FUNCTION fcProcentualReduction
VAR_INPUT
	rLAkt      	: REAL;
    rLR1       	: REAL;
    rLR2       	: REAL;
END_VAR
VAR_OUTPUT
	rOut		: REAL;
END_VAR
VAR
	ayLR		: ARRAY[0..1] OF REAL;
    rTemp		: REAL;
    iFor1		: INT;
END_VAR

(* Array clean *)
FOR iFor1 := 0 TO 1 DO 
    ayLR[iFor1] := 0.0;
END_FOR;
ayLR[0] := rLR1;
ayLR[1] := rLR2;
(* Sortieren *)
IF ayLR[0] < ayLR[1] THEN
    rTemp           := ayLR[1];
    ayLR[1]         := ayLR[0];     
    ayLR[0]         := rTemp;   
END_IF;
 
(* Berechnen *)
rOut := TO_REAL(rLAkt);
FOR iFor1 := 0 TO 1 DO 
    IF ayLR[iFor1] <> 0 THEN
        rOut := rOut - (( rOut / 100 ) * ayLR[iFor1]);
    ELSE
        EXIT;    
    END_IF;    
END_FOR;

END_FUNCTION

// 21 Interface/ITF_Superheat
INTERFACE ITF_Superheat EXTENDS __SYSTEM.IQueryInterface

{attribute 'monitoring' := 'variable'}
PROPERTY proAcknowleg : BOOL
GET
END_GET
END_PROPERTY

{attribute 'monitoring' := 'variable'}
PROPERTY proAvailable : BOOL
GET
END_GET
END_PROPERTY

{attribute 'monitoring' := 'variable'}
PROPERTY proLockDown : BOOL
GET
END_GET
END_PROPERTY

PROPERTY proIsError : BOOL
GET
END_GET
END_PROPERTY

PROPERTY proIsWarning : BOOL
GET
END_GET
END_PROPERTY

PROPERTY prorOnY : REAL
GET
END_GET
END_PROPERTY

PROPERTY prorLowSuperheatValue : REAL
GET
END_GET
END_PROPERTY

PROPERTY prorActÜberhitzung : REAL
GET
END_GET
END_PROPERTY

PROPERTY prorSollÜberhitzung : REAL
GET
END_GET
END_PROPERTY

PROPERTY p_scBase_fbxEnable : CtaSysConfig.ITF_DATATYPE
GET
END_GET
END_PROPERTY

PROPERTY p_scBase_EnAlarmVentOffen : CtaSysConfig.ITF_DATATYPE
GET
END_GET
END_PROPERTY

PROPERTY p_scBase_fbtDelayStartAlarm : CtaSysConfig.ITF_DATATYPE
GET
END_GET
END_PROPERTY

PROPERTY p_scInfluxDb_fbxEnable : CtaSysConfig.ITF_DATATYPE
GET
END_GET
END_PROPERTY

PROPERTY p_scLowSuperheat_fbrMin : CtaSysConfig.ITF_DATATYPE
GET
END_GET
END_PROPERTY

PROPERTY p_scLowSuperheat_fbxEnable : CtaSysConfig.ITF_DATATYPE
GET
END_GET
END_PROPERTY

PROPERTY p_scLowSuperheat_fbtDelayStartRegler : CtaSysConfig.ITF_DATATYPE
GET
END_GET
END_PROPERTY

PROPERTY p_scLowSuperheat_fbrMax : CtaSysConfig.ITF_DATATYPE
GET
END_GET
END_PROPERTY

PROPERTY p_scLowSuperheat_fbrMinÖffnung : CtaSysConfig.ITF_DATATYPE
GET
END_GET
END_PROPERTY

PROPERTY p_scLowSuperheat_fbxEnableWarning : CtaSysConfig.ITF_DATATYPE
GET
END_GET
END_PROPERTY

PROPERTY p_scLowSuperheat_fbxEnableAlarm : CtaSysConfig.ITF_DATATYPE
GET
END_GET
END_PROPERTY

PROPERTY p_scLowSuperheat_fbtDelayStartAlarm : CtaSysConfig.ITF_DATATYPE
GET
END_GET
END_PROPERTY

PROPERTY P_scLowSuperheat_fbrLowShAlarmValue : CtaSysConfig.ITF_REAL
GET
END_GET
END_PROPERTY

PROPERTY p_scMOP_fbxEnable : CtaSysConfig.ITF_DATATYPE
GET
END_GET
END_PROPERTY

PROPERTY p_scMOP_fbxEnableWarning : CtaSysConfig.ITF_DATATYPE
GET
END_GET
END_PROPERTY

PROPERTY p_scMOP_fbxEnableAlarm : CtaSysConfig.ITF_DATATYPE
GET
END_GET
END_PROPERTY

PROPERTY p_scMOP_fbtDelayStartAlarm : CtaSysConfig.ITF_DATATYPE
GET
END_GET
END_PROPERTY

PROPERTY p_scMOP_fbrMopSollwert : CtaSysConfig.ITF_DATATYPE
GET
END_GET
END_PROPERTY

PROPERTY proRefTofbPidSuperheat : REFERENCE TO CtaAppPid.fbPid
GET
END_GET
END_PROPERTY

PROPERTY proRefTofbSuperheatDumper : REFERENCE TO CtaAppDumper.fbDumper
GET
END_GET
END_PROPERTY

PROPERTY proRefTofbPidMop : REFERENCE TO CtaAppPid.fbPid
GET
END_GET
END_PROPERTY

PROPERTY proRefTofbMopDumper : REFERENCE TO CtaAppDumper.fbDumper
GET
END_GET
END_PROPERTY

{attribute 'hide'} 
PROPERTY INTERNAL proITF_REPORTMANAGER : CtaAppReport.ITF_REPORTMANAGER
GET
END_GET
END_PROPERTY

END_INTERFACE

// 40 Visualizations/VisSuperheat/visSuperheat
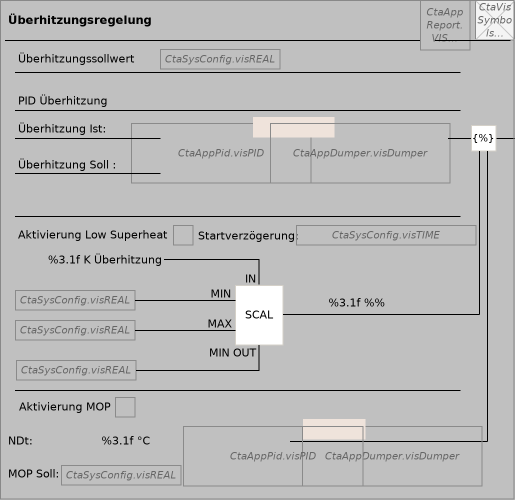
VISUALIZATION visSuperheat  // 515x500
VAR_INPUT
	ITF_SuperheatIN				: ITF_Superheat;
END_VAR
VAR_IN_OUT	
	fbrÜberhitzungssollwertIN 	: CtaSysConfig.fbREAL;	
END_VAR
    Frame (131,123 180x60)
        shows CtaAppPid.visPID(fbPID := ITF_SuperheatIN.proRefTofbPidSuperheat)
    Rectangle (253,117 81x20)
    Frame (270,123 180x60)
        shows CtaAppDumper.visDumper(fbDumper := ITF_SuperheatIN.proRefTofbSuperheatDumper)
    Line (448,138) (530,138)
    Label (5,10 200x20), "Überhitzungsregelung"
    Line (5,40) (420,40)
    Label (15,49 150x20), "Überhitzungssollwert"
    Frame (160,49 120x20)
        shows CtaSysConfig.visREAL(visfbREALIn := fbrÜberhitzungssollwertIN, stPhysikalischeEinheit := 'K')
    Label (15,119 120x20), "Überhitzung Ist:"
    Label (15,155 120x20), "Überhitzung Soll :"
    Textfield (471,125 25x26), "{%}"
    Frame (173,225 20x20)
        shows CtaSysConfig.visBOOL(visfbBOOLIn := ITF_SuperheatIN.p_scLowSuperheat_fbxEnable)
    Label (15,225 160x20), "Aktivierung Low Superheat"
    Label (195,226 120x20), "Startverzögerung:"
    Frame (296,225 180x20)
        shows CtaSysConfig.visTIME(visfbTIMEIn := ITF_SuperheatIN.p_scLowSuperheat_fbtDelayStartRegler)
    Line (15,216) (460,216)
    Line (15,390) (460,390)
    Label (16,397 100x20), "Aktivierung MOP"
    Frame (115,397 20x20)
        shows CtaSysConfig.visBOOL(visfbBOOLIn := ITF_SuperheatIN.p_scMOP_fbxEnable)
    Textfield (15,250 150x20), "%3.1f K Überhitzung", text variable: ITF_SuperheatIN.prorActÜberhitzung
    Frame (15,290 120x20)
        shows CtaSysConfig.visREAL(visfbREALIn := ITF_SuperheatIN.p_scLowSuperheat_fbrMin, stPhysikalischeEinheit := 'K')
    Frame (15,320 120x20)
        shows CtaSysConfig.visREAL(visfbREALIn := ITF_SuperheatIN.p_scLowSuperheat_fbrMax, stPhysikalischeEinheit := 'K')
    Frame (16,360 120x20)
        shows CtaSysConfig.visREAL(visfbREALIn := ITF_SuperheatIN.p_scLowSuperheat_fbrMinÖffnung, stPhysikalischeEinheit := '%')
    Line (15,72) (460,72)
    Line (15,138) (160,138)
    Line (15,173) (160,173)
    Textfield (235,285 48x60), "SCAL"
    Line (135,300) (235,300)
    Line (135,330) (235,330)
    Label (194,284 40x20), "MIN"
    Label (195,314 40x20), "MAX"
    Line (136,370) (259,370)
    Line (259,370) (259,345)
    Line (164,259) (259,259)
    Line (259,284) (259,259)
    Label (219,269 40x20), "IN"
    Label (201,343 58x20), "MIN OUT"
    Line (283,314) (479,314)
    Line (479,151) (479,314)
    Textfield (71,431 110x20), "%3.1f °C", text variable: ITF_SuperheatIN.prorActÜberhitzung
    Line (290,441) (487,441)
    Frame (302,426 180x60)
        shows CtaAppDumper.visDumper(fbDumper := ITF_SuperheatIN.proRefTofbMopDumper)
    Line (487,151) (487,441)
    Textfield (297,293 120x20), "%3.1f %%", text variable: ITF_SuperheatIN.prorLowSuperheatValue
    Image (475,0 40x40), image: CtaVisSymbols.ImagePool.gear
        OnMouseClick:  Dialog=PopUp, Parameters={uiPopUpGruppe: 1, ITF_SuperheatIN: ITF_SuperheatIN}, OpenModal=True, OpenCentered=True
    Frame (420,0 50x50)
        shows ReportIcon(ITF_REPORTMANAGER_IN := ITF_SuperheatIN.proITF_REPORTMANAGER)
        OnMouseClick:  Dialog=PopUp, Parameters={uiPopUpGruppe: 0, ITF_SuperheatIN: ITF_SuperheatIN}, OpenModal=True, OpenCentered=True
    Line (435,40) (510,40)
    Rectangle (303,419 62x20)
    Frame (183,426 180x60)
        shows CtaAppPid.visPID(fbPID := ITF_SuperheatIN.proRefTofbPidMop)
    Frame (61,465 120x20)
        shows CtaSysConfig.visREAL(visfbREALIn := ITF_SuperheatIN.p_scMOP_fbrMopSollwert, stPhysikalischeEinheit := '°c')
    Label (5,431 60x20), "NDt:"
    Label (5,464 60x20), "MOP Soll:"
    Label (15,91 150x20), "PID Überhitzung"
    Line (15,110) (460,110)
END_VISUALIZATION

// 40 Visualizations/Report/ReportIcon
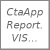
VISUALIZATION ReportIcon  // 50x50
VAR_INPUT
	ITF_REPORTMANAGER_IN	: CtaAppReport.ITF_REPORTMANAGER;
END_VAR
    Frame (0,0 50x50)
        shows CtaAppReport.VIS_ANZ_REPORTS_MODUL(ITF_REPORTMANAGER_IN := ITF_REPORTMANAGER_IN)
END_VISUALIZATION

// 40 Visualizations/Report/VIS_SUPERHEAT_REPORTS
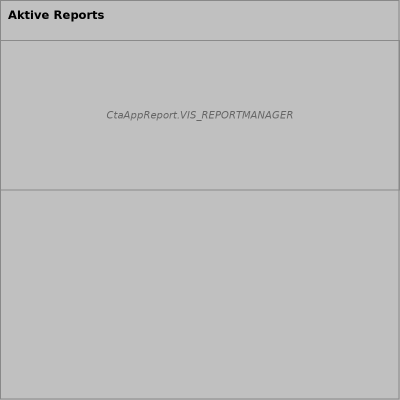
VISUALIZATION VIS_SUPERHEAT_REPORTS  // 400x400
VAR_INPUT
    ITF_SuperheatIN    :   ITF_Superheat;	
END_VAR
    Frame (0,40 400x150)
        shows CtaAppReport.VIS_REPORTMANAGER(ITF_REPORTMANAGER := ITF_SuperheatIN.proITF_REPORTMANAGER)
    Label (5,5 350x20), "Aktive Reports"
END_VISUALIZATION

// 40 Visualizations/PopUp/PopUp
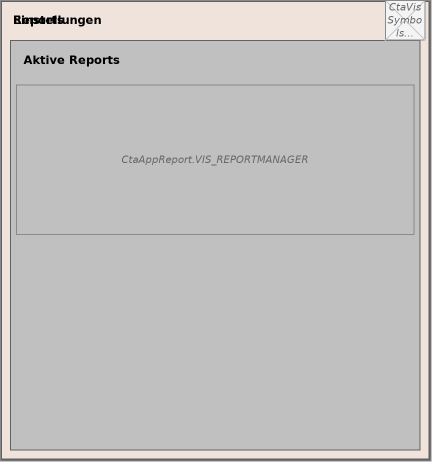
VISUALIZATION PopUp  // 432x462
VAR_INPUT
	ITF_SuperheatIN		: 	ITF_Superheat;
	uiPopUpGruppe		:	UINT;
END_VAR
    RoundedRectangle (0,0 430x460)
    RoundedRectangle (10,40 410x410)
    Image (385,0 40x40), image: CtaVisSymbols.ImagePool.close_solo_black
        OnMouseClick:  Dialog=PopUp, Result=None, NumpadKeypadSet=True
    Frame (16,45 398x399), frame switch variable: uiPopUpGruppe
        shows VIS_SUPERHEAT_REPORTS(ITF_SuperheatIN := ITF_SuperheatIN)
        shows VIS_SUPERHEAT_SETTINGS(ITF_SuperheatIN := ITF_SuperheatIN)
        pReferences[1]: ITF_ANTRIEBIN=ITF_SuperheatIN
    Label (10,0 150x40), "Reports", invisible if: uiPopUpGruppe = 1
    Label (10,0 150x40), "Einstellungen", invisible if: uiPopUpGruppe = 0
END_VISUALIZATION

// 40 Visualizations/Settings/VIS_SUPERHEAT_SETTINGS
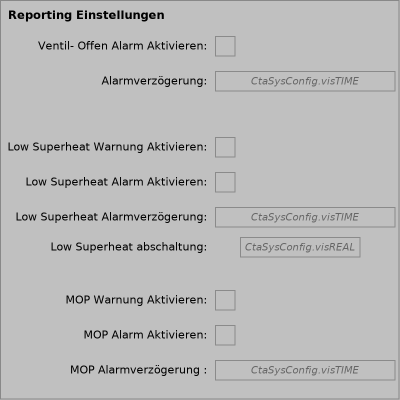
VISUALIZATION VIS_SUPERHEAT_SETTINGS  // 400x400
VAR_INPUT
    ITF_SuperheatIN    :   ITF_Superheat;	
END_VAR
    Frame (0,0 400x400)
        shows VIS_SUPERHEAT_SETTINGS_BASE(ITF_SuperheatIN := ITF_SuperheatIN)
END_VISUALIZATION

// 40 Visualizations/Settings/VIS_SUPERHEAT_SETTINGS_BASE
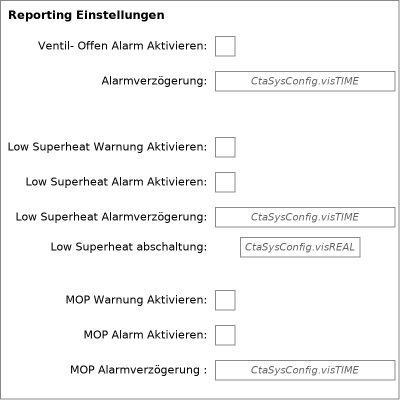
VISUALIZATION VIS_SUPERHEAT_SETTINGS_BASE  // 400x400
VAR_INPUT
    ITF_SuperheatIN    :   ITF_Superheat;	
END_VAR
    Label (5,5 350x20), "Reporting Einstellungen"
    Frame (215,36 20x20)
        shows CtaSysConfig.visBOOL(visfbBOOLIn := ITF_SuperheatIN.p_scBase_EnAlarmVentOffen)
    Label (10,36 200x20), "Ventil- Offen Alarm Aktivieren:"
    Frame (215,137 20x20)
        shows CtaSysConfig.visBOOL(visfbBOOLIn := ITF_SuperheatIN.p_scLowSuperheat_fbxEnableWarning)
    Label (10,137 200x20), "Low Superheat Warnung Aktivieren:"
    Frame (215,172 20x20)
        shows CtaSysConfig.visBOOL(visfbBOOLIn := ITF_SuperheatIN.p_scLowSuperheat_fbxEnableAlarm)
    Label (10,172 200x20), "Low Superheat Alarm Aktivieren:"
    Label (10,207 200x20), "Low Superheat Alarmverzögerung:"
    Label (10,290 200x20), "MOP Warnung Aktivieren:"
    Frame (215,71 180x20)
        shows CtaSysConfig.visTIME(visfbTIMEIn := ITF_SuperheatIN.p_scBase_fbtDelayStartAlarm)
    Label (10,325 200x20), "MOP Alarm Aktivieren:"
    Label (10,360 200x20), "MOP Alarmverzögerung :"
    Frame (215,360 180x20)
        shows CtaSysConfig.visTIME(visfbTIMEIn := ITF_SuperheatIN.p_scMOP_fbtDelayStartAlarm)
    Frame (215,290 20x20)
        shows CtaSysConfig.visBOOL(visfbBOOLIn := ITF_SuperheatIN.p_scMOP_fbxEnableWarning)
    Label (10,71 200x20), "Alarmverzögerung:"
    Frame (215,207 180x20)
        shows CtaSysConfig.visTIME(visfbTIMEIn := ITF_SuperheatIN.p_scLowSuperheat_fbtDelayStartAlarm)
    Frame (215,325 20x20)
        shows CtaSysConfig.visBOOL(visfbBOOLIn := ITF_SuperheatIN.p_scMOP_fbxEnableAlarm)
    Label (10,237 200x20), "Low Superheat abschaltung:"
    Frame (240,237 120x20)
        shows CtaSysConfig.visREAL(visfbREALIn := ITF_SuperheatIN.P_scLowSuperheat_fbrLowShAlarmValue, stPhysikalischeEinheit := 'K')
END_VISUALIZATION

(* text list Error (id | default | de)
  0 | Keine Meldung Anstehend | Keine Meldung Anstehend
  1 | Fehler Tiefe überhitzung | Fehler Tiefe überhitzung
  2 | MOP Fehler | MOP Fehler
  3 | Ventilöffnung zu Gross | Ventilöffnung zu Gross
  4 | Konfigurationsfehler speichern fehlgeschlagen reboot | Konfigurationsfehler speichern fehlgeschlagen reboot
   |  |  *)

(* text list Info (id | default)
   |  *)

(* text list Warnung (id | default | de)
  0 | Keine Meldung Anstehend | Keine Meldung Anstehend
  1 | Warnung Tiefe überhitzung | Warnung Tiefe überhitzung
  2 | Warnung MOP | Warnung MOP
   |  |  *)
